FUNCTION "LAxisCtrl_UnpubAxisPosition" : LReal
{ S7_Optimized_Access := 'TRUE' }
AUTHOR : 'tech.team.motioncontrol@siemens.com'
FAMILY : AxisCtrl
VERSION : 1.1
   VAR_INPUT
      axis : DB_ANY;
   END_VAR


BEGIN
	// Read axis parameter
	CASE TypeOfDB(#axis) OF
	  TO_PositioningAxis:
	    #LAxisCtrl_UnpubAxisPosition := "LAxisCtrl_UnpubPositionPosAxis"(#axis);

	  TO_SynchronousAxis:
	    #LAxisCtrl_UnpubAxisPosition := "LAxisCtrl_UnpubPositionSyncAxis"(#axis);

	  ELSE
	    #LAxisCtrl_UnpubAxisPosition := 0.0;
	END_CASE;
END_FUNCTION

